TYPE ST_KeyenceLaser_Block_Edit_Request_Completion_Clear :
STRUCT
Character_String_Setting_Read_Complete_Clear		: BIT;
Character_String_Printed_Read_Complete_Clear		: BIT;
Character_String_Change_Complete_Clear				: BIT;
Reserve_0											: BIT;
Reserve_1											: BIT;
Reserve_2											: BIT;
Reserve_3											: BIT;
Reserve_4											: BIT;
END_STRUCT
END_TYPE

(* stored: Version 1.1.0.1, ProductVersion 3.1.4024.11
   DUT ST_KeyenceLaser_Block_Edit_Request_Completion_Clear: Id {eefab645-1573-44df-92f0-bf65ffa31d24} *)
